KUKA KRL program: PontoAjuste.src, PontoAjuste.dat

--- PontoAjuste.src ---
&ACCESS RVO
&REL 6
DEF  PontoAjuste ( )
   ;FOLD INI;%{PE}
      ;FOLD BASISTECH INI
         GLOBAL INTERRUPT DECL 3 WHEN $STOPMESS==TRUE DO IR_STOPM ( )
         INTERRUPT ON 3
         BAS (#INITMOV,0 )
      ;ENDFOLD (BASISTECH INI)
      ;FOLD USER INI
         ;Make your modifications here
         $TOOL = TOOL_DATA[1]
         $BASE = $NULLFRAME
      ;ENDFOLD (USER INI)
   ;ENDFOLD (INI)

   ;FOLD PTP HOME  Vel= 100 % DEFAULT;%{PE}%MKUKATPBASIS,%CMOVE,%VPTP,%P 1:PTP, 2:HOME, 3:, 5:100, 7:DEFAULT
      $BWDSTART = FALSE
      PDAT_ACT=PDEFAULT
      FDAT_ACT=FHOME
      BAS (#PTP_PARAMS,100 )
      $H_POS=XHOME
      PTP  XHOME
   ;ENDFOLD

   ;ALINHE BEM A GARRA COM A ESTEIRA
   ;TOUCHUP ESTEIRA 1
   ;FOLD PTP XServiceEsteira1 Vel=100 % PDAT2 Tool[1]:GarraUniversal Base[0];%{PE}
      ;FOLD Parameters ;%{h}
         ;Params IlfProvider=kukaroboter.basistech.inlineforms.movement.old; Kuka.IsGlobalPoint=False; Kuka.PointName=xservice; Kuka.BlendingEnabled=False; Kuka.MoveDataPtpName=PDAT2; Kuka.VelocityPtp=100; Kuka.CurrentCDSetIndex=0; Kuka.MovementParameterFieldEnabled=True; IlfCommand=PTP
      ;ENDFOLD
      $BWDSTART = FALSE
      PDAT_ACT = PPDATSS
      FDAT_ACT = Fxservice
      BAS(#PTP_PARAMS, 100.0)
      SET_CD_PARAMS (0)
      PTP XServiceEsteira1 C_DIS
   ;ENDFOLD

   ;TOUCHUP ESTEIRA 2
   ;FOLD PTP XServiceEsteira2 Vel=100 % PDAT2 Tool[1]:GarraUniversal Base[0];%{PE}
      ;FOLD Parameters ;%{h}
         ;Params IlfProvider=kukaroboter.basistech.inlineforms.movement.old; Kuka.IsGlobalPoint=False; Kuka.PointName=xservice; Kuka.BlendingEnabled=False; Kuka.MoveDataPtpName=PDAT2; Kuka.VelocityPtp=100; Kuka.CurrentCDSetIndex=0; Kuka.MovementParameterFieldEnabled=True; IlfCommand=PTP
      ;ENDFOLD
      $BWDSTART = FALSE
      PDAT_ACT = PPDATSS
      FDAT_ACT = Fxservice
      BAS(#PTP_PARAMS, 100.0)
      SET_CD_PARAMS (0)
      PTP XServiceEsteira2 C_DIS
   ;ENDFOLD

   ;ALINHE BEM A GARRA COM O PALLET

   ;TOUCHUP PALLET 1
   ;FOLD PTP XServicePallet1 Vel=100 % PDAT2 Tool[1]:GarraUniversal Base[0];%{PE}
      ;FOLD Parameters ;%{h}
         ;Params IlfProvider=kukaroboter.basistech.inlineforms.movement.old; Kuka.IsGlobalPoint=False; Kuka.PointName=xservice; Kuka.BlendingEnabled=False; Kuka.MoveDataPtpName=PDAT2; Kuka.VelocityPtp=100; Kuka.CurrentCDSetIndex=0; Kuka.MovementParameterFieldEnabled=True; IlfCommand=PTP
      ;ENDFOLD
      $BWDSTART = FALSE
      PDAT_ACT = PPDATSS
      FDAT_ACT = Fxservice
      BAS(#PTP_PARAMS, 100.0)
      SET_CD_PARAMS (0)
      PTP XServicePallet1 C_DIS
   ;ENDFOLD

   ;TOUCHUP PALLET 2
   ;FOLD PTP XServicePallet2 Vel=100 % PDAT2 Tool[1]:GarraUniversal Base[0];%{PE}
      ;FOLD Parameters ;%{h}
         ;Params IlfProvider=kukaroboter.basistech.inlineforms.movement.old; Kuka.IsGlobalPoint=False; Kuka.PointName=xservice; Kuka.BlendingEnabled=False; Kuka.MoveDataPtpName=PDAT2; Kuka.VelocityPtp=100; Kuka.CurrentCDSetIndex=0; Kuka.MovementParameterFieldEnabled=True; IlfCommand=PTP
      ;ENDFOLD
      $BWDSTART = FALSE
      PDAT_ACT = PPDATSS
      FDAT_ACT = Fxservice
      BAS(#PTP_PARAMS, 100.0)
      SET_CD_PARAMS (0)
      PTP XServicePallet2 C_DIS
   ;ENDFOLD

   ;ATUALIZA OFFSETS
   ;AtualizaOffsets( )

   ;ADICIONE AQUI PONTOS DA SUA ESCOLHA



   ;###################################

   ;FOLD PTP HOME  Vel= 100 % DEFAULT;%{PE}%MKUKATPBASIS,%CMOVE,%VPTP,%P 1:PTP, 2:HOME, 3:, 5:100, 7:DEFAULT
      $BWDSTART = FALSE
      PDAT_ACT=PDEFAULT
      FDAT_ACT=FHOME
      BAS (#PTP_PARAMS,100 )
      $H_POS=XHOME
      PTP  XHOME
   ;ENDFOLD
END

--- PontoAjuste.dat ---
&ACCESS RVO
&REL 6
DEFDAT  PONTOAJUSTE PUBLIC
;FOLD EXTERNAL DECLARATIONS;%{PE}%MKUKATPBASIS,%CEXT,%VCOMMON,%P
;FOLD BASISTECH EXT;%{PE}%MKUKATPBASIS,%CEXT,%VEXT,%P
EXT  BAS (BAS_COMMAND  :IN,REAL  :IN )
;ENDFOLD (BASISTECH EXT)
;FOLD USER EXT;%{E}%MKUKATPUSER,%CEXT,%VEXT,%P
;Make your modifications here

;pontos exportados de FURUKAWA
DECL PDAT PPDAT1G={VEL 100.000,ACC 100.000,APO_DIST 500.000,APO_MODE #CDIS,GEAR_JERK 100.000,EXAX_IGN 0}
DECL LDAT LCPDAT1G={VEL 2.00000,ACC 100.000,APO_DIST 500.000,APO_FAC 50.0000,AXIS_VEL 100.000,AXIS_ACC 100.000,ORI_TYP #VAR,CIRC_TYP #BASE,JERK_FAC 50.0000,GEAR_JERK 100.000,EXAX_IGN 0}
DECL FDAT FP1G={TOOL_NO 0,BASE_NO 0,IPO_FRAME #BASE,POINT2[] " "}

;PONTOS SERVICE GLOBAL

DECL GLOBAL E6POS XServiceEsteira1={X 2099.77441,Y 445.740936,Z -7.67726088,A -179.925095,B 8.91580273E-15,C 180.000,S 2,T 35,E1 0.0,E2 0.0,E3 0.0,E4 0.0,E5 0.0,E6 0.0}
DECL GLOBAL E6POS XServiceEsteira2={X 2099.77441,Y 445.740936,Z -7.67726088,A -179.925095,B 8.91580273E-15,C 180.000,S 2,T 35,E1 0.0,E2 0.0,E3 0.0,E4 0.0,E5 0.0,E6 0.0}

DECL GLOBAL E6POS XServicePallet1={X 2099.77441,Y 445.740936,Z -7.67726088,A -179.925095,B 8.91580273E-15,C 180.000,S 2,T 35,E1 0.0,E2 0.0,E3 0.0,E4 0.0,E5 0.0,E6 0.0}
DECL GLOBAL E6POS XServicePallet2={X 2099.77441,Y 445.740936,Z -7.67726088,A -179.925095,B 8.91580273E-15,C 180.000,S 2,T 35,E1 0.0,E2 0.0,E3 0.0,E4 0.0,E5 0.0,E6 0.0}

;------ OUTROS PONTOS ------


;ENDFOLD (USER EXT)
;ENDFOLD (EXTERNAL DECLARATIONS)
DECL MODULEPARAM_T LAST_TP_PARAMS={PARAMS[] "Kuka.PointName=xservice; Kuka.FrameData.base_no=0; Kuka.FrameData.tool_no=1; Kuka.FrameData.ipo_frame=#BASE; Kuka.isglobalpoint=False; Kuka.MoveDataPtpName=PDAT2; Kuka.MovementDataPdat.apo_mode=#CDIS; Kuka.MovementDataPdat.apo_dist=500; Kuka.MovementData.vel=100; Kuka.MovementData.acc=100; Kuka.MovementData.gear_jerk=100; Kuka.MovementData.exax_ign=0; Kuka.VelocityPtp=100; Kuka.BlendingEnabled=False; Kuka.CurrentCDSetIndex=0"}
DECL FDAT Fxservice={TOOL_NO 1,BASE_NO 0,IPO_FRAME #BASE,POINT2[] " "}
DECL PDAT PPDATSS={VEL 100.000,ACC 100.000,APO_DIST 500.000,APO_MODE #CDIS,GEAR_JERK 100.000,EXAX_IGN 0}
DECL E6POS Xxservice={X 2099.77441,Y 445.740936,Z -7.67726088,A -179.925095,B 8.91580273E-15,C 180.000,S 2,T 35,E1 0.0,E2 0.0,E3 0.0,E4 0.0,E5 0.0,E6 0.0}
ENDDAT
